FUNCTION_BLOCK E_DELAY (* Delayed event propagation *)
  (* Standard: 61499-1 Annex A; Description: Copyright (c) 2017 fortiss GmbH This program and the accompanying materials are made available under the terms of the Eclipse Public License 2.0 which is available at https://www.eclipse.org/legal/epl-2.0/ SPDX-License-Identifier: EPL-2.0 *)
  (* Version 1.0, 2017-09-21, Alois Zoitl, fortiss GmbH, initial API and implementation and/or initial documentation *)
  (* Version 3.0, 2025-04-14, Patrick Aigner, changed package *)
  PACKAGE iec61499::events;
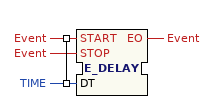
  EVENT_INPUT
    START WITH DT; (* Start delayed event propagation *)
    STOP; (* Stop the delayed event propagation *)
  END_EVENT
  EVENT_OUTPUT
    EO; (* Delayed event *)
  END_EVENT
  VAR_INPUT
    DT : TIME; (* Delay time, >0 *)
  END_VAR
  (* Service APPLICATION/RESOURCE: Delayed event propagation *)
END_FUNCTION_BLOCK
